FUNCTION_BLOCK Motor_Enable
VAR_INPUT
	Disable_motor: BOOL;
	DesiredSpeedPWM:INT;
	PositiveDirection: BOOL;
	NegativeDirection: BOOL;
END_VAR
VAR_OUTPUT
	setEnable: INT;
	setSpeedPWM:INT; 
END_VAR
VAR
	move_enabled: BOOL;
END_VAR
VAR // added by the converter: edge detectors and wires of the graphical bodies
    _w1, _w2 : BOOL;
END_VAR

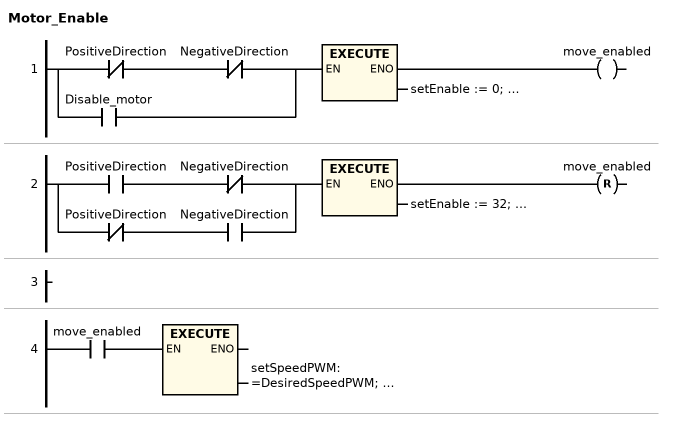
// NETWORK 1
_w1 := NOT PositiveDirection AND NOT NegativeDirection OR Disable_motor;
IF _w1 THEN
    setEnable := 0;
    setSpeedPWM:=0;
END_IF
move_enabled := _w1;

// NETWORK 2
_w2 := PositiveDirection AND NOT NegativeDirection OR NOT PositiveDirection AND NegativeDirection;
IF _w2 THEN setEnable := 32; END_IF
move_enabled R= _w2;

// NETWORK 3

// NETWORK 4
IF move_enabled THEN setSpeedPWM:=DesiredSpeedPWM; END_IF

END_FUNCTION_BLOCK

(* stored: Version 1.1.0.1, ProductVersion 3.1.4024.12
   POU Motor_Enable: Id {6b1b4b10-fbd2-4184-b8c1-f01bb9c7c68a}, SpecialFunc None *)
